FUNCTION_BLOCK ThreeConCtl (* Composite Function Block Type *)
  (* Standard: 61499-2 *)
  (* Version 0.2, 2003-12-05, JHC, Rockwell Automation, Renamed from NEWCOMPFB. *)
  (* Version 0.1, 2002-01-08, JHC, Rockwell Automation, Added DLY FB as example. *)
  (* Version 0.0, 2000-05-27, JHC, Rockwell Automation *)
  (* Compiler header: package fb.rt.cs725; *)
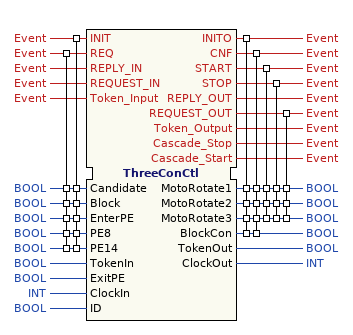
  EVENT_INPUT
    INIT WITH Candidate, Block, EnterPE, PE8, PE14; (* Initialization Request *)
    REQ WITH Block, Candidate, EnterPE, PE8, PE14; (* Normal Execution Request *)
    REPLY_IN;
    REQUEST_IN;
    Token_Input;
  END_EVENT
  EVENT_OUTPUT
    INITO WITH MotoRotate1, MotoRotate2, MotoRotate3, BlockCon; (* Initialization Confirm *)
    CNF WITH MotoRotate1, MotoRotate2, MotoRotate3, BlockCon; (* Execution Confirmation *)
    START WITH MotoRotate1, MotoRotate2, MotoRotate3;
    STOP WITH MotoRotate1, MotoRotate2, MotoRotate3;
    REPLY_OUT;
    REQUEST_OUT WITH MotoRotate1, MotoRotate2, MotoRotate3;
    Token_Output;
    Cascade_Stop;
    Cascade_Start;
  END_EVENT
  VAR_INPUT
    Candidate : BOOL;
    Block : BOOL;
    EnterPE : BOOL;
    PE8 : BOOL;
    PE14 : BOOL;
    TokenIn : BOOL;
    ExitPE : BOOL;
    ClockIn : INT;
    ID : BOOL;
  END_VAR
  VAR_OUTPUT
    MotoRotate1 : BOOL;
    MotoRotate2 : BOOL;
    MotoRotate3 : BOOL;
    BlockCon : BOOL;
    TokenOut : BOOL;
    ClockOut : INT;
  END_VAR
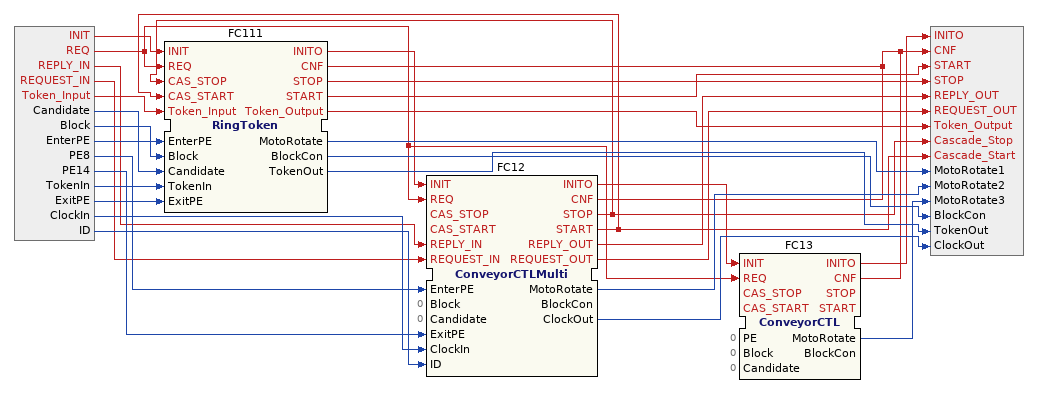
  FBS
    FC12 : ConveyorCTLMulti(Block := 0, Candidate := 0);
    FC13 : ConveyorCTL(Block := 0, Candidate := 0, PE := 0);
    FC111 : RingToken;
  END_FBS
  EVENT_CONNECTIONS
    FC12.INITO TO FC13.INIT;
    FC13.INITO TO INITO;
    FC13.CNF TO CNF;
    REQ TO FC12.REQ;
    REQ TO FC13.REQ;
    FC12.CNF TO CNF;
    REPLY_IN TO FC12.REPLY_IN;
    REQUEST_IN TO FC12.REQUEST_IN;
    FC12.REQUEST_OUT TO REQUEST_OUT;
    FC12.REPLY_OUT TO REPLY_OUT;
    FC12.STOP TO Cascade_Stop;
    FC12.START TO Cascade_Start;
    FC111.CNF TO CNF;
    FC111.STOP TO STOP;
    FC111.START TO START;
    FC111.Token_Output TO Token_Output;
    Token_Input TO FC111.Token_Input;
    REQ TO FC111.REQ;
    INIT TO FC111.INIT;
    FC111.INITO TO FC12.INIT;
    FC12.STOP TO FC111.CAS_STOP;
    FC12.START TO FC111.CAS_START;
  END_CONNECTIONS
  DATA_CONNECTIONS
    FC13.MotoRotate TO MotoRotate3;
    FC12.MotoRotate TO MotoRotate2;
    EnterPE TO FC111.EnterPE;
    Block TO FC111.Block;
    Candidate TO FC111.Candidate;
    TokenIn TO FC111.TokenIn;
    ExitPE TO FC111.ExitPE;
    FC111.MotoRotate TO MotoRotate1;
    FC111.BlockCon TO BlockCon;
    FC111.TokenOut TO TokenOut;
    PE8 TO FC12.EnterPE;
    PE14 TO FC12.ExitPE;
    ID TO FC12.ID;
    ClockIn TO FC12.ClockIn;
    FC12.ClockOut TO ClockOut;
  END_CONNECTIONS
END_FUNCTION_BLOCK
